// TIA Portal V16 export
// export: Created 2024-09-05T17:40:15.2765473Z, ExportSetting WithDefaults, DisplayName Totally Integrated Automation Portal, DisplayVersion V16 Update 6, DisplayName TIA Portal Version Control Interface, DisplayVersion V16 Update 2, DisplayName TIA Portal Openness, DisplayVersion V16 Update 6, DisplayName STEP 7 Professional, DisplayVersion V16 Update 6, DisplayName STEP 7 Safety, DisplayVersion V16, DisplayName WinCC Advanced, DisplayVersion V16 Update 6
TYPE "connectionParameterType"
// stored: IsFailsafeCompliant false
   STRUCT
      ConnectInfo { ExternalAccessible := 'False'; ExternalVisible := 'False'; ExternalWritable := 'False'; S7_SetPoint := 'True'} : OPC_UA_SessionConnectInfo;
      ConnectionHdl { ExternalAccessible := 'False'; ExternalVisible := 'False'; ExternalWritable := 'False'} : DWord := 16#0;
      ServerEndpointUrl { ExternalAccessible := 'False'; ExternalVisible := 'False'; ExternalWritable := 'False'} : String[254] := 'opc.tcp://192.168.0.2:4840';
   END_STRUCT;
   // ConnectInfo.SessionName := WSTRING#'OPC UA Connection_1';
   // ConnectInfo.ApplicationName := WSTRING#'';
   // ConnectInfo.SecurityMsgMode := 1;
   // ConnectInfo.SecurityPolicy := 1;
   // ConnectInfo.ServerUri := '';
   // ConnectInfo.CheckServerCertificate := False;
   // ConnectInfo.TransportProfile := 1;
   // ConnectInfo.UserIdentityTokenType := 0;
   // ConnectInfo.UserTokenParam1 := WSTRING#'';
   // ConnectInfo.UserTokenParam2 := WSTRING#'';
   // ConnectInfo.CertificateID := 0;
   // ConnectInfo.SessionTimeout := T#30S;
   // ConnectInfo.MonitorConnection := T#5S;
   // ConnectInfo.LocaleIDs[0] := 'en-US';
   // ConnectInfo.LocaleIDs[1..4] := '';
END_TYPE
